(* Logix 5000 project; controller IPG_2332_07A 1769-L16ER-BB1B rev 34.12; software revision 34.01 *)

TASK MAIN_10Ms (periodic, rate 10 ms, priority 1, watchdog 500 ms) : MainProgram_10Ms
TASK MainTask (continuous, watchdog 500 ms) : MainProgram

MODULES
   Local : 1769-L16ER-BB1B (PointIO 0, rev 34.12)
      VS_063 : EX260-SEN1 (Ethernet 192.168.0.63, rev 1.1, Output RPI 10 ms)
      Camera_065 : vendor 678 type 100 code 274 (Ethernet 192.168.0.65, rev 11.1, Output RPI 60 ms)
      QR_064 : vendor 678 type 773 code 1330 (Ethernet 192.168.0.64, rev 1.6, StandardDataDriven RPI 20 ms)
           QR_064:I1.Data[3].4   // QR Results Valid
           QR_064:I1.Data[0].3   // MIssed Trigger
           QR_064:I1.Data[1]   // Results Status
           QR_064:I1.Data[6]   // Trigger Count
           QR_064:I1.Data[1].0   // Results Available
           QR_064:I1.Data[1].7   // General Fault
           QR_064:I1.Data[1].1   // Result Ack Mirror
           QR_064:I1.Data[2].6   // QR Trigger Ack
           QR_064:I1.Data[0].6   // Trigger IN1-Pin4 Current State
           QR_064:I1.Data[0].2   // Aquiring
           QR_064:I1.Data[0].4   // Current Mode (0- Setup Tool Mode, 1- Run Mode)
           QR_064:I1.Data[8]   // Result Count
           QR_064:I1.Data[0].0   // Trigger Ready
           QR_064:I1.Data[0].1   // Trigger Ack
           QR_064:I1.Data[0].5   // Serial Error (0- no error or in configuration mode, 1 - No Reader connected)
           QR_064:I1.Data[1].2   // Result Data Buffer Overrun
           QR_064:I1.Data[0]   // Trigger Status
           QR_064:I1.Data[0].7   // Trigger IN2-Pin2 Current State
           QR_064:O1.Data[0].1   // Trigger
           QR_064:O1.Data[0].0   // Trigger Enable
           QR_064:O1.Data[0].5   // QR Trigger
      Discrete_IO : Embedded (PointIO 1, rev 34.11, Output RPI 20 ms)
      C_ANALOG_01 : 1734-OE2V (PointIO 3, rev 3.1, Output RPI 80 ms)
      RS232 : 1734-232ASC (PointIO 2, rev 4.1, Output RPI 80 ms)
      C_ANALOG_02 : 1734-OE2V (PointIO 4, rev 3.1, Output RPI 80 ms)
END_MODULES

TYPE DateTime :
STRUCT
   Year : DINT;
   Month : DINT;
   Day : DINT;
   Hour : DINT;
   Minute : DINT;
   Second : DINT;
   MicroSecond : DINT;
END_STRUCT
END_TYPE

TYPE String_1 :
STRUCT
   LEN : DINT;
   DATA : SINT[1];
END_STRUCT
END_TYPE

TYPE String_15 :
STRUCT
   LEN : DINT;
   DATA : SINT[15];
END_STRUCT
END_TYPE

TYPE String_60 :
STRUCT
   LEN : DINT;
   DATA : SINT[60];
END_STRUCT
END_TYPE

TYPE udt_Controller_Status :
STRUCT
   Battery_Status : BOOL;
   Forces_Installed : BOOL;
   Forces_Enabled : BOOL;
   Controller_Mode : DINT;   // 1 = Program 2= Run 3 = Remote Run 4= Remote Test 5 = Remote Program 6 = Fault
   Controller_Status : DINT;
   Device_Status : DINT;
   Fault_Status : DINT;
   Forces_Status : DINT;   // 0 = No Forces, Forces not Enabled 1 = Forces Enabled 2 = Forces Installed
   IO_Status : DINT;   // 0 = LED Off 1 = Flashing Red 2 = Flashing Green 3 = Solid Green
   Key_Switch_Status : DINT;   // 1 = Run 2 = Program 3 = Remote
   Minor_Fault : DINT;
END_STRUCT
END_TYPE

TYPE udt_HMI_IO_Desc :
STRUCT
   Increment_Page : BOOL;
   Increment_Event : BOOL;
   Increment_OS : BOOL;
   Decrement_Page : BOOL;
   Decrement_Event : BOOL;
   Decrement_OS : BOOL;
   Two_Column_Display : BOOL;   // On = 2 Column Display
   Index : DINT;
   Max_Index : DINT;   // Maximum Index
   Status : INT[2];
   IO_Desc : udt_IO_Desc[16];
END_STRUCT
END_TYPE

TYPE udt_HMI_Message :
STRUCT
   Message : String_60;
   Background : DINT;
END_STRUCT
END_TYPE

TYPE udt_HMI_Message_Display :
STRUCT
   Message : udt_HMI_Message;
   Index : DINT;
END_STRUCT
END_TYPE

TYPE udt_HMI_Optix :
STRUCT
   Current_Display_Name : STRING;
   Previous_Display_Name : STRING;
   Project_Name : STRING;
   Active_Language : String_15;
   Heartbeat : BOOL;
END_STRUCT
END_TYPE

TYPE udt_HMI_PB :
STRUCT
   PB : DINT;
   ONS : DINT;
   PB_OS : DINT;
END_STRUCT
END_TYPE

TYPE udt_IO_Desc :
STRUCT
   Address : STRING_16;
   Description : STRING_32;
END_STRUCT
END_TYPE

TYPE udt_LED :
STRUCT
   Max_Voltage : INT;
   Ramp_Timer : TIMER;
   On_Timer : TIMER;
   Voltage_Out : INT;
   Delay_Timer : TIMER;
   On_Time : REAL;
   Delay_Time : REAL;
   Ramp_Time : REAL;
END_STRUCT
END_TYPE

TYPE udt_Machine_Control_V2 :
STRUCT
   Alarm : BOOL;
   Alarm_Silence : BOOL;
   Auto_Mode : BOOL;
   Auto_On_OS : BOOL;
   Auto_Off_OS : BOOL;
   Conveyors_Run : BOOL;
   Conveyors_Running : BOOL;
   Conveyors_On_OS : BOOL;
   Conveyors_Off_OS : BOOL;
   Conveyor_Stop_Req : BOOL;
   Conveyor_Stop : BOOL;
   Cycle_Enable : BOOL;   // Cycle Enable
   Fault_Reset : BOOL;   // Reset Fault
   Guard_Closed : BOOL;
   Master_Reset : BOOL;   // Master Reset
   Pwr_Up_Chk : BOOL;   // Power up Light check
   Pwr_On : BOOL;   // Power On
   Reset : BOOL;   // Reset
   Reset_Counts : BOOL;
   Safety_OK : BOOL;   // Safety Ok
   Reset_OS : BOOL;
   Single_Cycle : BOOL;   // Single Cycle
   Single_Cycle_On_OS : BOOL;
   Single_Cycle_Off_OS : BOOL;
   Stop : BOOL;   // Stop Position
   Stop_Pos : BOOL;
   Stop_Req : BOOL;   // Stop Request
   Update_OS : BOOL;   // Update Results
   Start_OS : BOOL;
   Sequence_Reset : BOOL;   // Reset Sequence
   Alarm_Monitor : BOOL[32];   // Alarm Monitor Conditions
   Reset_Cnt : COUNTER;   // Reset Counter
   HMI_Mode_Display : DINT;   // HMI Mode Display
   HMI_PB : udt_HMI_PB;   // HMI Pushbuttons
   Message_Index : DINT;   // MMI Message Index
   OS : DINT;   // one shots
   Counts : DINT[3];   // Station Production Counts
   Conveyor_Start_Dly : TIMER;   // Conveyor Start Delay
   Guard_Close_Delay : TIMER;
   Guard_Unlock_Dly : TIMER;
   Guard_Unlock_Timer : TIMER;
   Pwr_On_Dly : TIMER;   // Power On Delay Timer
   Safety_Ok_Dly : TIMER;   // Safety Ok Delay
   Reset_Duration : TIMER;   // Reset Duration
   Cycle_Time : TIMER;
   Conveyor_Speed : REAL;
END_STRUCT
END_TYPE

TYPE udt_Shift_Register :
STRUCT
   SR : DINT;   // Shift Register
   Part_Style : DINT;   // Part Style
   Height : REAL;   // Height
END_STRUCT
END_TYPE

TYPE udt_Station_Sequence :
STRUCT
   Done : BOOL;   // Sequence Done/Complete
   Home : BOOL;   // Station Home
   In_Process : BOOL;   // Sequence In Process
   Request : BOOL;   // Sequence Request
   Position : DINT;
   OS : DINT;
   OS1 : DINT;
   OS2 : DINT;
   StepOS : DINT;
   StepOS1 : DINT;
   StepOS2 : DINT;
   Timer : TIMER[20];
   Result : BOOL;   // 0=Fail, 1=Pass
END_STRUCT
END_TYPE

TYPE udt_Zaber_Axis :
STRUCT
   Home : BOOL;
   InPos : BOOL;
   ActPos_Step_String : STRING;
   CmdPos_mm : REAL;
   CmdPos_Step_Dint : DINT;
   CmdPos_Step_String : STRING;
   Write_String : STRING;
   Read_String : STRING;
   Write : SERIAL_PORT_CONTROL;
   MoveReq : BOOL;
   Reset : BOOL;
   Home_String : STRING; {access Read Only}
   MovAbs_String : STRING;
   MovAbs : BOOL;
   Return_String : STRING;
   MovRel_String : STRING;
   MovRel : BOOL;
   Resloution : REAL;   // micrometers per step
   Manual_MovAbs : BOOL;
   Jog_Fwd : BOOL;
   Jog_Fwd_String : STRING;
   Jog_Rev : BOOL;
   Jog_Rev_String : STRING;
   Jog_Value_mm : REAL;
   Go_Home : BOOL;
   Go_CmdPos : BOOL;
   Jog_Value_Step_Dint : DINT;
   Jog_Value_Step_String : STRING;
   Store_CmdPos : BOOL;
   Get_Pos_String : STRING;
   Store_CmdPos_Delay : TIMER;
   String_Pos_Found : DINT;
   String_Pos_Length : DINT;
   Get_Pos : BOOL;
   WriteReq : BOOL;
   Status : STRING;
   Moving : BOOL;
   Idle : STRING;
   IdlePos : DINT;
   Zero : STRING;
   Get_Pos_Delay : TIMER;
   Busy : STRING;
   BusyPos : DINT;
   Axis_String : STRING;
   Axis_Dint : DINT;
   HMI_PB : udt_HMI_PB;
   Store_CmdPos_Reset_Delay : TIMER;
   ActPos_Step_Dint : DINT;
   ActPos_mm : REAL;
   Reset_String : STRING;
END_STRUCT
END_TYPE

ADD_ON_INSTRUCTION AOI_Convert_hhmmss   (* revision 1.0 *)
VAR_INPUT
   Hour : DINT; {required}
   Minutes : DINT; {required}
   Seconds : DINT; {required}
END_VAR
VAR_IN_OUT
   Time : String_15; {required}
END_VAR
VAR
   String_Hour : String_15; {access None}
   String_Minute : String_15; {access None}
   String_Seconds : String_15; {access None}
   String_Colon : String_1 := ':'; {access None}
   Temp_String : String_15; {access None}
   String_Zero : String_1 := '0'; {access None}
END_VAR

ROUTINE Logic   (* ladder *)
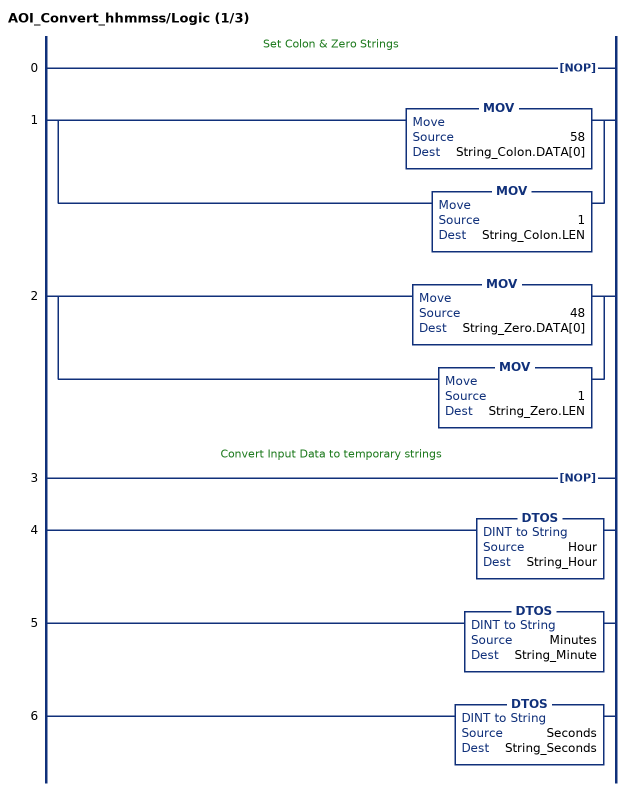
   // Set Colon & Zero Strings
   0: NOP();
   1: [MOV(58,String_Colon.DATA[0]) ,MOV(1,String_Colon.LEN) ];
   2: [MOV(48,String_Zero.DATA[0]) ,MOV(1,String_Zero.LEN) ];
   // Convert Input Data to temporary strings
   3: NOP();
   4: DTOS(Hour,String_Hour);
   5: DTOS(Minutes,String_Minute);
   6: DTOS(Seconds,String_Seconds);
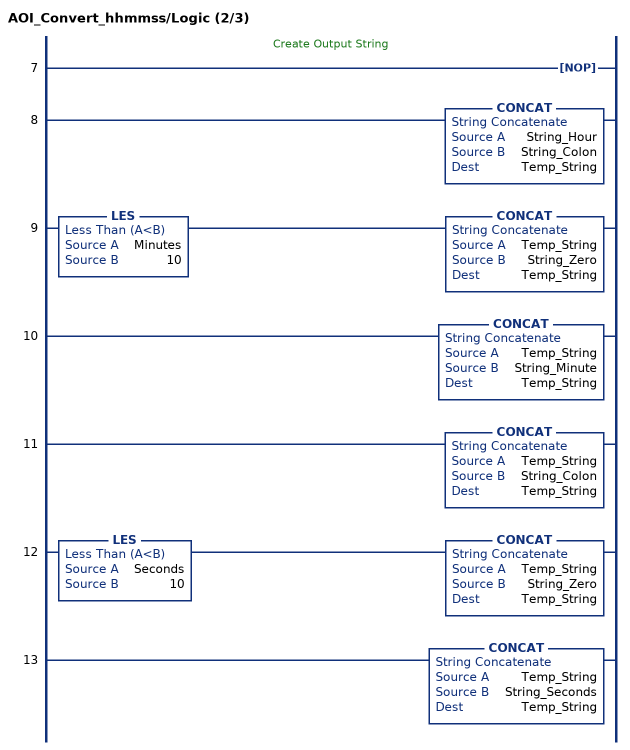
   // Create Output String
   7: NOP();
   8: CONCAT(String_Hour,String_Colon,Temp_String);
   9: LES(Minutes,10)CONCAT(Temp_String,String_Zero,Temp_String);
   10: CONCAT(Temp_String,String_Minute,Temp_String);
   11: CONCAT(Temp_String,String_Colon,Temp_String);
   12: LES(Seconds,10)CONCAT(Temp_String,String_Zero,Temp_String);
   13: CONCAT(Temp_String,String_Seconds,Temp_String);
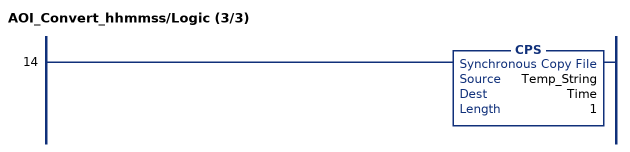
   14: CPS(Temp_String,Time,1);
END_ROUTINE
END_ADD_ON_INSTRUCTION

ADD_ON_INSTRUCTION AOI_Cycle_Times   (* revision 1.0 *)
VAR_INPUT
   Start_Timing_IN : BOOL; {visible}
   In_Process_IN : BOOL; {visible}
   Alarmed_IN : BOOL; {visible}
   Waiting_IN : BOOL; {visible}
   Update_IN : BOOL; {visible}
   Uptime_IN : BOOL; {visible}
   Downtime_IN : BOOL; {visible}
   Data_Reset_IN : BOOL; {visible}
END_VAR
VAR_OUTPUT
   Avg_Cycle_Time : REAL; {access Read Only, visible}
   Cycle_Time : REAL; {access Read Only, visible}
   Avg_PTP_Cycle_Time : REAL; {access Read Only, visible}
   Part_Part_Cycle_Time : REAL; {access Read Only, visible}
END_VAR
VAR_INPUT
   Current_Cycle : REAL; {visible}
END_VAR
VAR_IN_OUT
   Waiting_Time : String_15; {required}
   Alarmed_Time : String_15; {required}
   Uptime_Time : String_15; {required}
   Downtime_Time : String_15; {required}
END_VAR
VAR
   p_Timer : TIMER := (PRE := 100); {access None}
   p_Accumulated_mS : DINT; {access None}
   p_ONS : DINT; {access None}
   p_Start_Time_mS : DINT; {access None}
   p_End_Time_mS : DINT; {access None}
   p_Cycle_Time_mS : DINT; {access None}
   p_Total_Cycles : DINT; {access None}
   p_Avg_PTP_Cycle_Time_Raw : DINT; {access None}
   p_Waiting_Accumulated_mS : DINT; {access None}
   p_Convert_Waiting_AOI : AOI_Convert_hhmmss; {access None}
   p_Convert_Alarmed_AOI : AOI_Convert_hhmmss; {access None}
   p_Avg_Cycle_Time_Raw : DINT; {access None}
   p_Uptime_mSeconds : DINT; {access None}
   p_Uptime_Seconds : DINT; {access None}
   p_Uptime_Minutes : DINT; {access None}
   p_Uptime_Hours : DINT; {access None}
   p_Convert_Uptime_AOI : AOI_Convert_hhmmss; {access None}
   p_Waiting_Hours : DINT; {access Read Only}
   p_Waiting_Minutes : DINT; {access Read Only}
   p_Waiting_Seconds : DINT; {access Read Only}
   p_Alarm_Hours : DINT; {access Read Only}
   p_Alarm_Minutes : DINT; {access Read Only}
   p_Alarm_mSeconds : DINT; {access None}
   p_Alarm_Seconds : DINT; {access Read Only}
   p_Convert_Downtime_AOI : AOI_Convert_hhmmss; {access None}
   p_Downtime_Hours : DINT; {access None}
   p_Downtime_Minutes : DINT; {access None}
   p_Downtime_Seconds : DINT; {access None}
   p_Downtime_mSeconds : DINT; {access None}
END_VAR

ROUTINE Logic   (* ladder *)
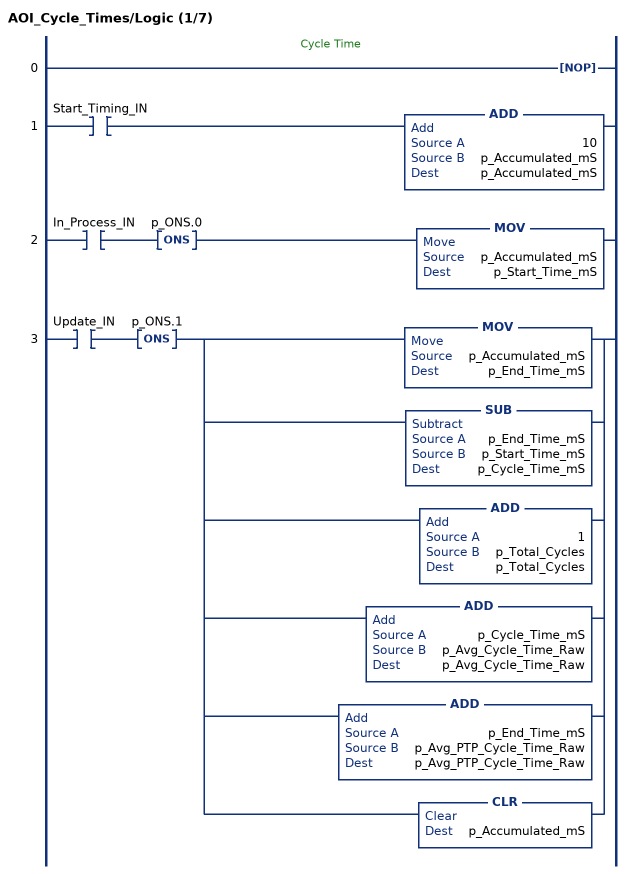
   // Cycle Time
   0: NOP();
   1: XIC(Start_Timing_IN)ADD(10,p_Accumulated_mS,p_Accumulated_mS);
   2: XIC(In_Process_IN)ONS(p_ONS.0)MOV(p_Accumulated_mS,p_Start_Time_mS);
   3: XIC(Update_IN)ONS(p_ONS.1)[MOV(p_Accumulated_mS,p_End_Time_mS) ,SUB(p_End_Time_mS,p_Start_Time_mS,p_Cycle_Time_mS) ,ADD(1,p_Total_Cycles,p_Total_Cycles) ,ADD(p_Cycle_Time_mS,p_Avg_Cycle_Time_Raw,p_Avg_Cycle_Time_Raw) ,ADD(p_End_Time_mS,p_Avg_PTP_Cycle_Time_Raw,p_Avg_PTP_Cycle_Time_Raw) ,CLR(p_Accumulated_mS) ];
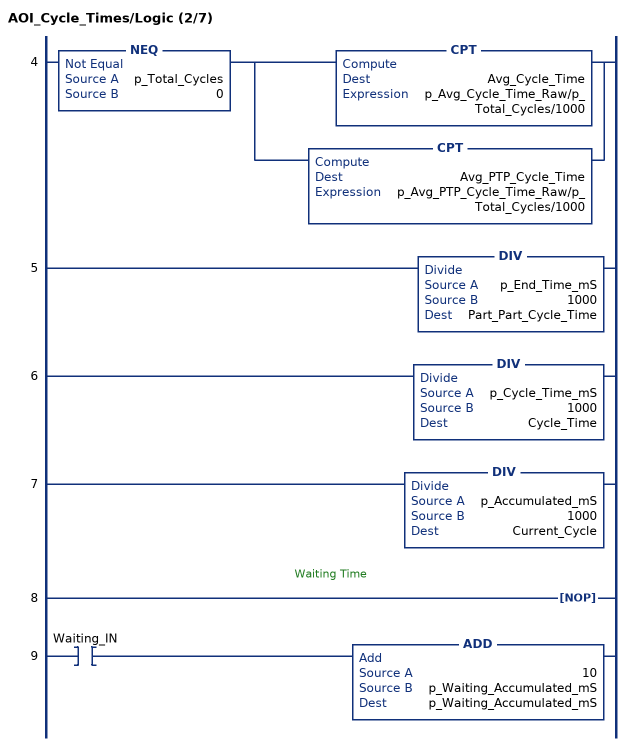
   4: NEQ(p_Total_Cycles,0)[CPT(Avg_Cycle_Time,p_Avg_Cycle_Time_Raw/p_Total_Cycles/1000) ,CPT(Avg_PTP_Cycle_Time,p_Avg_PTP_Cycle_Time_Raw/p_Total_Cycles/1000) ];
   5: DIV(p_End_Time_mS,1000,Part_Part_Cycle_Time);
   6: DIV(p_Cycle_Time_mS,1000,Cycle_Time);
   7: DIV(p_Accumulated_mS,1000,Current_Cycle);
   // Waiting Time
   8: NOP();
   9: XIC(Waiting_IN)ADD(10,p_Waiting_Accumulated_mS,p_Waiting_Accumulated_mS);
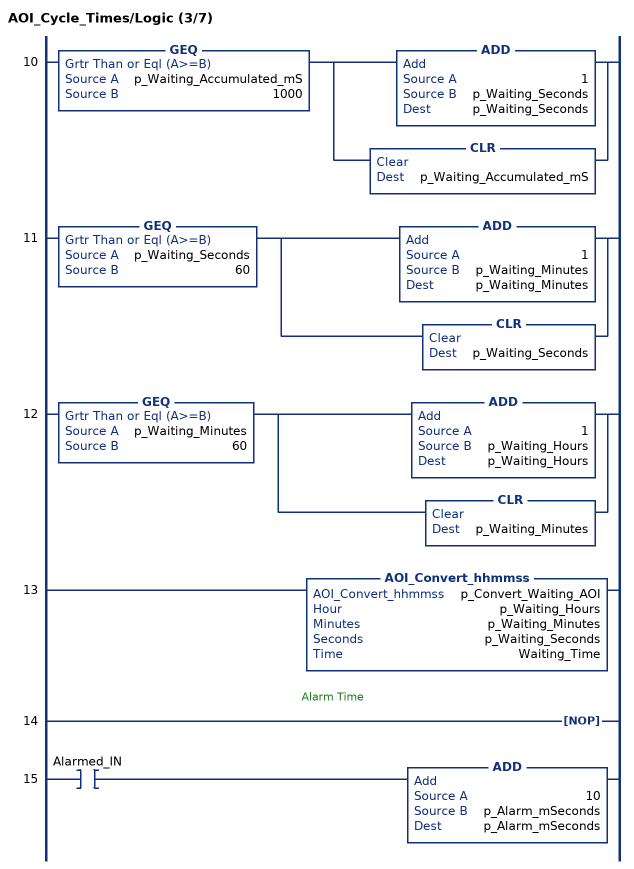
   10: GEQ(p_Waiting_Accumulated_mS,1000)[ADD(1,p_Waiting_Seconds,p_Waiting_Seconds) ,CLR(p_Waiting_Accumulated_mS) ];
   11: GEQ(p_Waiting_Seconds,60)[ADD(1,p_Waiting_Minutes,p_Waiting_Minutes) ,CLR(p_Waiting_Seconds) ];
   12: GEQ(p_Waiting_Minutes,60)[ADD(1,p_Waiting_Hours,p_Waiting_Hours) ,CLR(p_Waiting_Minutes) ];
   13: AOI_Convert_hhmmss(p_Convert_Waiting_AOI,p_Waiting_Hours,p_Waiting_Minutes,p_Waiting_Seconds,Waiting_Time);
   // Alarm Time
   14: NOP();
   15: XIC(Alarmed_IN)ADD(10,p_Alarm_mSeconds,p_Alarm_mSeconds);
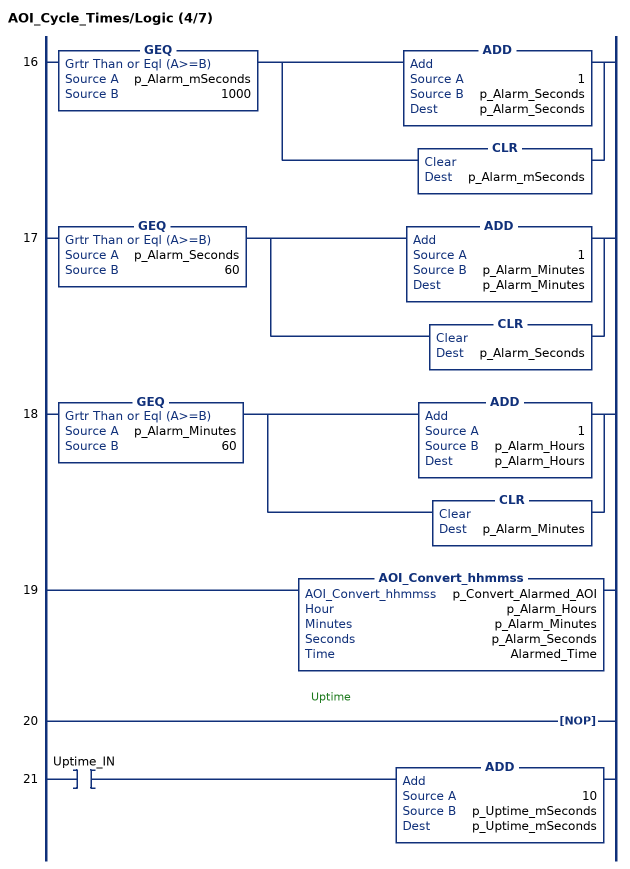
   16: GEQ(p_Alarm_mSeconds,1000)[ADD(1,p_Alarm_Seconds,p_Alarm_Seconds) ,CLR(p_Alarm_mSeconds) ];
   17: GEQ(p_Alarm_Seconds,60)[ADD(1,p_Alarm_Minutes,p_Alarm_Minutes) ,CLR(p_Alarm_Seconds) ];
   18: GEQ(p_Alarm_Minutes,60)[ADD(1,p_Alarm_Hours,p_Alarm_Hours) ,CLR(p_Alarm_Minutes) ];
   19: AOI_Convert_hhmmss(p_Convert_Alarmed_AOI,p_Alarm_Hours,p_Alarm_Minutes,p_Alarm_Seconds,Alarmed_Time);
   // Uptime
   20: NOP();
   21: XIC(Uptime_IN)ADD(10,p_Uptime_mSeconds,p_Uptime_mSeconds);
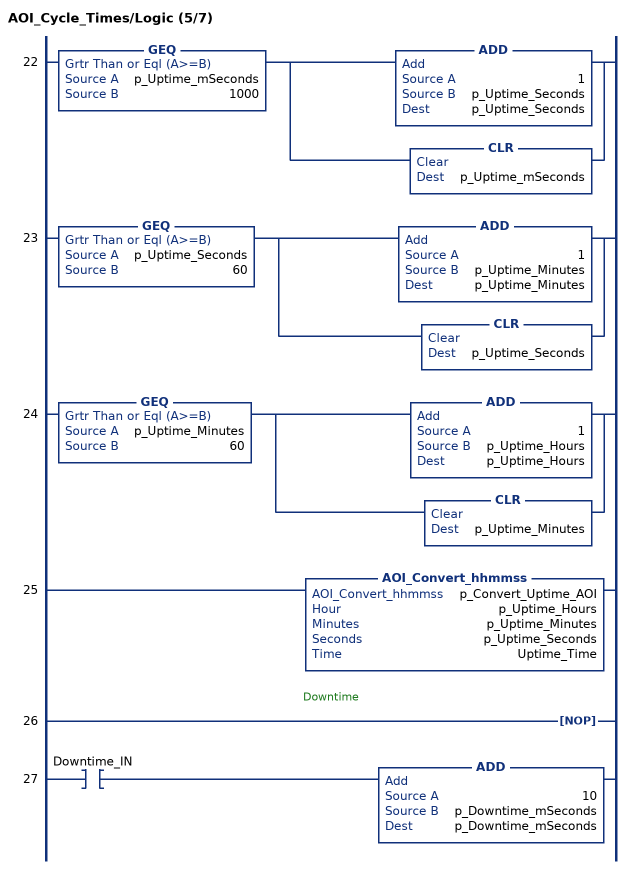
   22: GEQ(p_Uptime_mSeconds,1000)[ADD(1,p_Uptime_Seconds,p_Uptime_Seconds) ,CLR(p_Uptime_mSeconds) ];
   23: GEQ(p_Uptime_Seconds,60)[ADD(1,p_Uptime_Minutes,p_Uptime_Minutes) ,CLR(p_Uptime_Seconds) ];
   24: GEQ(p_Uptime_Minutes,60)[ADD(1,p_Uptime_Hours,p_Uptime_Hours) ,CLR(p_Uptime_Minutes) ];
   25: AOI_Convert_hhmmss(p_Convert_Uptime_AOI,p_Uptime_Hours,p_Uptime_Minutes,p_Uptime_Seconds,Uptime_Time);
   // Downtime
   26: NOP();
   27: XIC(Downtime_IN)ADD(10,p_Downtime_mSeconds,p_Downtime_mSeconds);
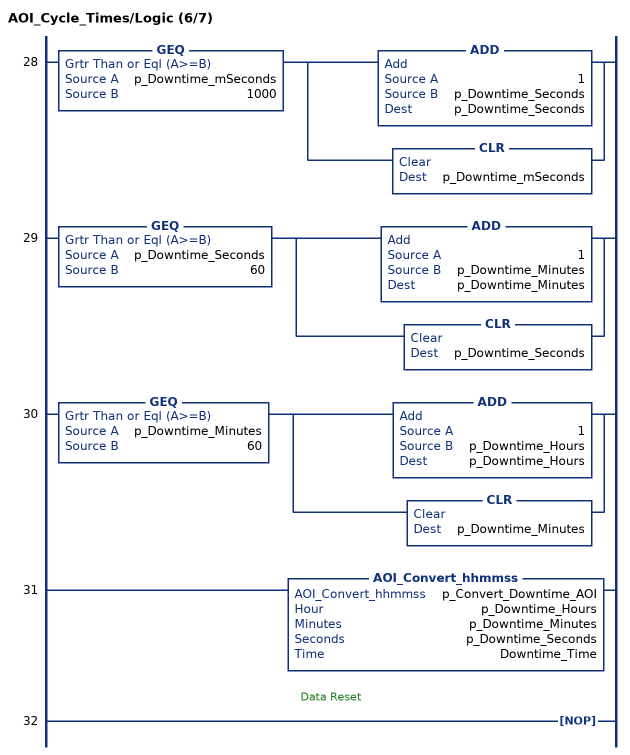
   28: GEQ(p_Downtime_mSeconds,1000)[ADD(1,p_Downtime_Seconds,p_Downtime_Seconds) ,CLR(p_Downtime_mSeconds) ];
   29: GEQ(p_Downtime_Seconds,60)[ADD(1,p_Downtime_Minutes,p_Downtime_Minutes) ,CLR(p_Downtime_Seconds) ];
   30: GEQ(p_Downtime_Minutes,60)[ADD(1,p_Downtime_Hours,p_Downtime_Hours) ,CLR(p_Downtime_Minutes) ];
   31: AOI_Convert_hhmmss(p_Convert_Downtime_AOI,p_Downtime_Hours,p_Downtime_Minutes,p_Downtime_Seconds,Downtime_Time);
   // Data Reset
   32: NOP();
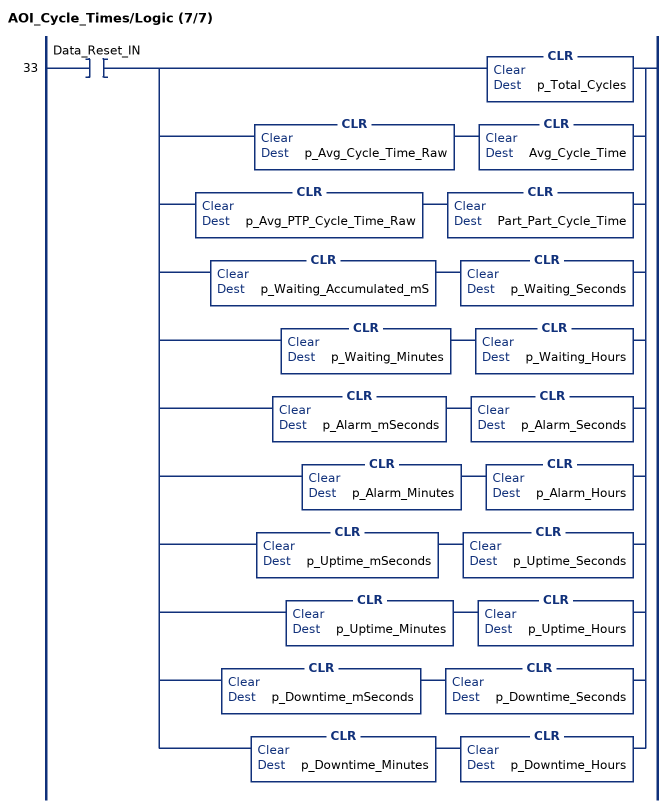
   33: XIC(Data_Reset_IN)[CLR(p_Total_Cycles) ,CLR(p_Avg_Cycle_Time_Raw) CLR(Avg_Cycle_Time) ,CLR(p_Avg_PTP_Cycle_Time_Raw) CLR(Part_Part_Cycle_Time) ,CLR(p_Waiting_Accumulated_mS) CLR(p_Waiting_Seconds) ,CLR(p_Waiting_Minutes) CLR(p_Waiting_Hours) ,CLR(p_Alarm_mSeconds) CLR(p_Alarm_Seconds) ,CLR(p_Alarm_Minutes) CLR(p_Alarm_Hours) ,CLR(p_Uptime_mSeconds) CLR(p_Uptime_Seconds) ,CLR(p_Uptime_Minutes) CLR(p_Uptime_Hours) ,CLR(p_Downtime_mSeconds) CLR(p_Downtime_Seconds) ,CLR(p_Downtime_Minutes) CLR(p_Downtime_Hours) ];
END_ROUTINE
END_ADD_ON_INSTRUCTION

ADD_ON_INSTRUCTION AOI_PB_Confirm   (* revision 1.0 *)
VAR_INPUT
   Pushbutton_IN : BOOL; {required}
END_VAR
VAR_OUTPUT
   Confirmed_OUT : BOOL; {access Read Only, visible}
   State_OUT : DINT; {access Read Only, visible}
END_VAR
VAR
   PB_ONS : BOOL; {access None}
   Confirm_CTU : COUNTER := (PRE := 2); {access None}
   Confirm_Timeout : TIMER := (PRE := 2000); {access None}
   Confirmed_ONS : BOOL; {access None}
END_VAR

ROUTINE Logic   (* ladder *)
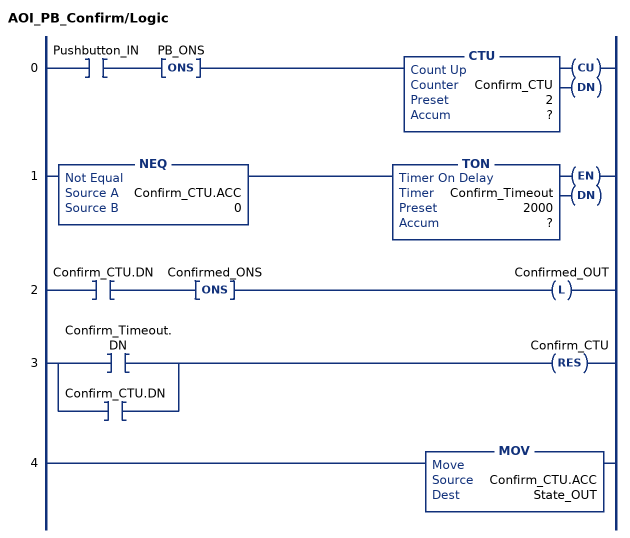
   0: XIC(Pushbutton_IN)ONS(PB_ONS)CTU(Confirm_CTU,?,?);
   1: NEQ(Confirm_CTU.ACC,0)TON(Confirm_Timeout,?,?);
   2: XIC(Confirm_CTU.DN)ONS(Confirmed_ONS)OTL(Confirmed_OUT);
   3: [XIC(Confirm_Timeout.DN) ,XIC(Confirm_CTU.DN) ]RES(Confirm_CTU);
   4: MOV(Confirm_CTU.ACC,State_OUT);
END_ROUTINE
END_ADD_ON_INSTRUCTION

ADD_ON_INSTRUCTION AOI_PLC_Status   (* revision 1.0 *)
VAR_IN_OUT
   HMI_PLC_Status : udt_Controller_Status; {required}
END_VAR

ROUTINE Logic   (* ladder *)
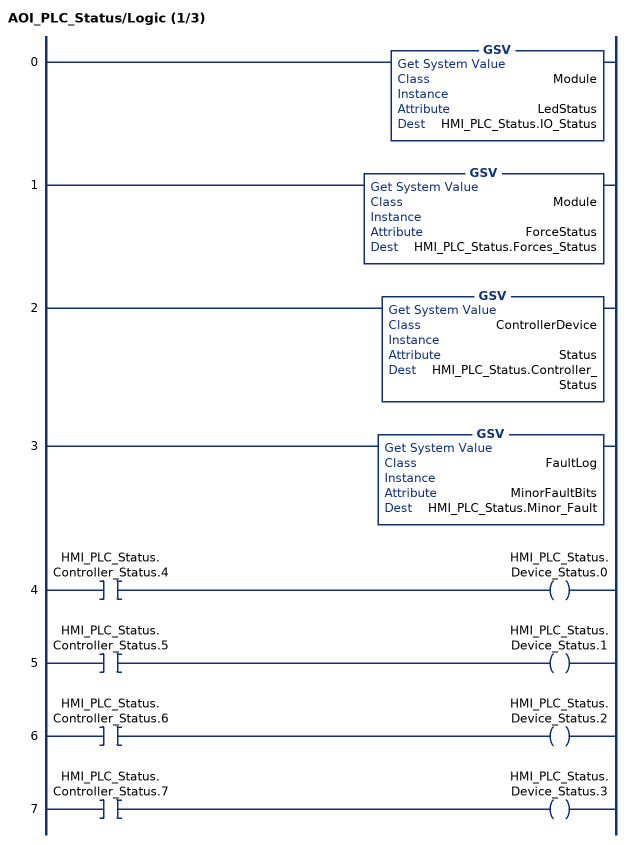
   0: GSV(Module,,LedStatus,HMI_PLC_Status.IO_Status);
   1: GSV(Module,,ForceStatus,HMI_PLC_Status.Forces_Status);
   2: GSV(ControllerDevice,,Status,HMI_PLC_Status.Controller_Status);
   3: GSV(FaultLog,,MinorFaultBits,HMI_PLC_Status.Minor_Fault);
   4: XIC(HMI_PLC_Status.Controller_Status.4)OTE(HMI_PLC_Status.Device_Status.0);
   5: XIC(HMI_PLC_Status.Controller_Status.5)OTE(HMI_PLC_Status.Device_Status.1);
   6: XIC(HMI_PLC_Status.Controller_Status.6)OTE(HMI_PLC_Status.Device_Status.2);
   7: XIC(HMI_PLC_Status.Controller_Status.7)OTE(HMI_PLC_Status.Device_Status.3);
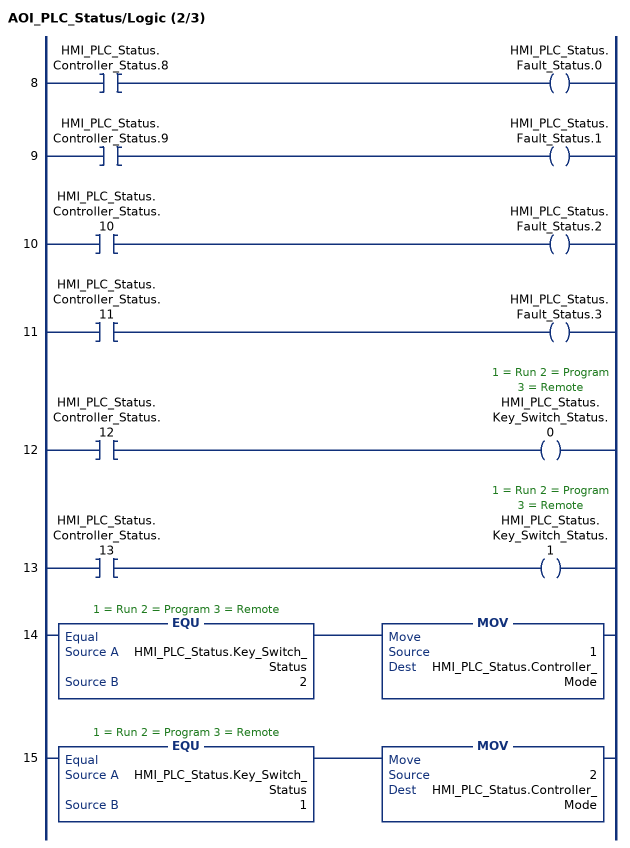
   8: XIC(HMI_PLC_Status.Controller_Status.8)OTE(HMI_PLC_Status.Fault_Status.0);
   9: XIC(HMI_PLC_Status.Controller_Status.9)OTE(HMI_PLC_Status.Fault_Status.1);
   10: XIC(HMI_PLC_Status.Controller_Status.10)OTE(HMI_PLC_Status.Fault_Status.2);
   11: XIC(HMI_PLC_Status.Controller_Status.11)OTE(HMI_PLC_Status.Fault_Status.3);
   12: XIC(HMI_PLC_Status.Controller_Status.12)OTE(HMI_PLC_Status.Key_Switch_Status.0);
   13: XIC(HMI_PLC_Status.Controller_Status.13)OTE(HMI_PLC_Status.Key_Switch_Status.1);
   14: EQU(HMI_PLC_Status.Key_Switch_Status,2)MOV(1,HMI_PLC_Status.Controller_Mode);
   15: EQU(HMI_PLC_Status.Key_Switch_Status,1)MOV(2,HMI_PLC_Status.Controller_Mode);
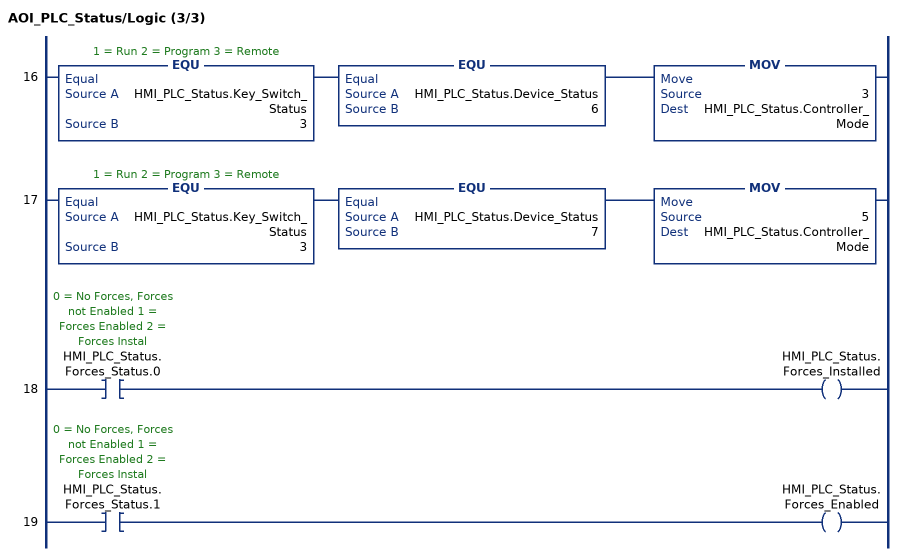
   16: EQU(HMI_PLC_Status.Key_Switch_Status,3)EQU(HMI_PLC_Status.Device_Status,6)MOV(3,HMI_PLC_Status.Controller_Mode);
   17: EQU(HMI_PLC_Status.Key_Switch_Status,3)EQU(HMI_PLC_Status.Device_Status,7)MOV(5,HMI_PLC_Status.Controller_Mode);
   18: XIC(HMI_PLC_Status.Forces_Status.0)OTE(HMI_PLC_Status.Forces_Installed);
   19: XIC(HMI_PLC_Status.Forces_Status.1)OTE(HMI_PLC_Status.Forces_Enabled);
END_ROUTINE
END_ADD_ON_INSTRUCTION

VAR_GLOBAL   (* controller tags *)
   DateTime : DateTime := (Year := 2023, Month := 12, Day := 8, Hour := 12, Minute := 11, Second := 26, MicroSecond := 594656);
   Debug_SDF : DINT := 64;
   HMI_IO_Description : udt_IO_Desc[96] := ([0].Address := 'Loc:I:1.0', [0].Description := 'E-Stop Relay Monitor', [1].Address := 'Loc:I:1.1', [1].Description := 'E-Stop PB', [2].Address := 'Loc:I:1.2', [2].Description := 'Door Safety Relay Monitor', [3].Address := 'Loc:I:1.3', [3].Description := 'Main Air Okay', [4].Address := 'Loc:I:1.4', [4].Description := 'Start PB', [5].Address := 'Loc:I:1.5', [5].Description := 'Spare', [6].Address := 'Loc:I:1.6', [6].Description := 'Spare', [7].Address := 'Loc:I:1.7', [7].Description := 'Spare', [8].Address := 'Loc:I:1.8', [8].Description := 'Ferrule Gripper Vac', [9].Address := 'Loc:I:1.9', [9].Description := 'Fiber Gripper Vac', [10].Address := 'Loc:I:1.10', [10].Description := 'Cassette Gripper Release', [11].Address := 'Loc:I:1.11', [11].Description := 'Cassette Gripper Extend', [12].Address := 'Loc:I:1.12', [12].Description := 'Cassette Gripper Retract', [13].Address := 'Loc:I:1.13', [13].Description := 'Cassette Presence', [14].Address := 'Loc:I:1.14', [14].Description := 'Spare', [15].Address := 'Loc:I:1.15', [15].Description := 'Spare', [16].Address := 'Loc:O:1.0', [16].Description := 'E-Stop Safety Reset', [17].Address := 'Loc:O:1.1', [17].Description := 'Spare', [18].Address := 'Loc:O:1.2', [18].Description := 'Light Stack Read', [19].Address := 'Loc:O:1.3', [19].Description := 'Light Stack Amber', [20].Address := 'Loc:O:1.4', [20].Description := 'Light Stack Green', [21].Address := 'Loc:O:1.5', [21].Description := 'Ferrule Gripper Solenoid', [22].Address := 'Loc:O:1.6', [22].Description := 'Fiber Gripper Solenoid', [23].Address := 'Loc:O:1.7', [23].Description := 'Spare', [24].Address := 'Loc:O:1.8', [24].Description := 'Dispenser Start', [25].Address := 'Loc:O:1.9', [25].Description := 'PB Light Red', [26].Address := 'Loc:O:1.10', [26].Description := 'PB Light Amber', [27].Address := 'Loc:O:1.11', [27].Description := 'PB Light Green', [28].Address := 'Loc:O:1.12', [28].Description := 'Work Light', [29].Address := 'Loc:O:1.13', [29].Description := 'Spare',
        [30].Address := 'Loc:O:1.14', [30].Description := 'Spare', [31].Address := 'Loc:O:1.15', [31].Description := 'Spare', [32].Address := 'VS_063:O:0.0', [32].Description := 'Cassette Release');
   HMI_Messages : udt_HMI_Message_Display[48] := ([1].Message.Message := 'Emergency Stop', [1].Message.Background := 1, [2].Message.Background := 1, [3].Message.Background := 1, [4].Message.Background := 1, [5].Message.Background := 1, [6].Message.Background := 1, [7].Message.Background := 1, [8].Message.Background := 1, [9].Message.Background := 1, [10].Message.Background := 1, [11].Message.Background := 1, [12].Message.Background := 1, [13].Message.Background := 1, [14].Message.Background := 1, [15].Message.Background := 1, [16].Message.Message := 'Safety Reset Required', [16].Message.Background := 6, [17].Message.Message := 'Machine Powering Up', [17].Message.Background := 4, [18].Message.Background := 4, [19].Message.Background := 3, [20].Message.Background := 3, [21].Message.Background := 3, [22].Message.Background := 3, [23].Message.Background := 3, [24].Message.Background := 3, [25].Message.Background := 3, [26].Message.Background := 3, [27].Message.Background := 3, [28].Message.Background := 3, [29].Message.Background := 3, [30].Message.Background := 3, [35].Message.Message := 'Machine Idle', [36].Message.Message := 'Machine Alarmed', [36].Message.Background := 1, [37].Message.Message := 'Machine Running', [37].Message.Background := 2, [41].Message.Message := 'Machine Stop Requested', [41].Message.Background := 2, [42].Message.Message := 'Machine in Setup/Step Mode', [42].Message.Background := 4, [44].Message.Message := 'Cycle Stop in Progress');
   HMI_Messages_Sequence : udt_HMI_Message_Display[20] := ([0].Message.Message := 'Idle', [1].Message.Message := 'Waiting for Cassette', [1].Message.Background := 4, [2].Message.Message := 'Fiber Vacuum On', [2].Message.Background := 2, [3].Message.Message := 'Ferrule Vacuum On', [3].Message.Background := 2, [4].Message.Message := 'Read Database', [4].Message.Background := 2, [5].Message.Message := 'Check Database', [5].Message.Background := 2, [6].Message.Message := 'Fiber Axis Down', [6].Message.Background := 2, [7].Message.Message := 'Syringe Axis In', [7].Message.Background := 2, [8].Message.Message := 'Dispense Glue', [8].Message.Background := 2, [9].Message.Message := 'Syringe Axis Out', [9].Message.Background := 2, [10].Message.Message := 'Mirror Axis In', [10].Message.Background := 2, [11].Message.Message := 'LED On', [11].Message.Background := 2, [12].Message.Message := 'Mirror Axis Out', [12].Message.Background := 2, [13].Message.Message := 'Ferrule Vacuum Off', [13].Message.Background := 2, [14].Message.Message := 'Fiber Axis Up', [14].Message.Background := 2, [15].Message.Message := 'Fiber Vacuum Off', [15].Message.Background := 2, [16].Message.Message := 'Sequence Complete', [16].Message.Background := 2, [17].Message.Background := 2, [18].Message.Background := 2, [19].Message.Background := 2);
END_VAR

PROGRAM MainProgram   (* main routine MainRoutine *)

ROUTINE MainRoutine   (* ladder *)
END_ROUTINE
END_PROGRAM

PROGRAM MainProgram_10Ms   (* main routine A_Main *)
VAR
   Axis_Controller : udt_Zaber_Axis := (Write_String := '/1 3 get pos$0D', Read_String := '$0A@01 3 OK IDLE -- 0$0D', Write.LEN := -243409016, Write.POS := -2147483640, Write.ERROR := 16#8000_0008, Home_String := '$C1$00$1C$00$01$00$00$00$00$00$00$00$00$00$00$00$08$00$00$80L$00$00$80$CCt9$F1$04<$00$00$9C$84$1B$00$14$01$00$00$02$00$00$00$00$00$00$00$01$00$00$00$00$00$00$00$00$00$00$00$00$00$00$00$00$00$00$00$00$00$00$00$00$00$00$00$00$00$00$00$00$00$00$00', Resloution := 8.e-45, Manual_MovAbs := 1, Jog_Rev_String := ' ', Go_CmdPos := 1, Jog_Value_Step_Dint := 32, Get_Pos_String := '$01$00$00$00$00$00$00$00$00$00$00$00$08$00$00$80$08$00$00$80$CCt9$F1$8C>$00$00$C1$00$15$00$01$00$00$00$00$00$00$00$18$00$08$80$08$00$00$80$08$00$00$80$CCt9$F1$AC>$00$00$C1$00$14$00$01$00$00$00$00$00$00$00$F4$01$00$00$08$00$00$80$08$00$00$80', Store_CmdPos_Delay.PRE := 16076, Store_CmdPos_Delay.ACC := 1245377, Store_CmdPos_Delay.EN := 1, Store_CmdPos_Delay.TT := 1, Store_CmdPos_Delay.DN := 1, String_Pos_Found := 1, Status := '$08$00$00$80$CCt9$F1$EC>$00$00$C1$00$12$00$01$00$00$00$00$00$00$00$00$00$00$00$08$00$00$80$08$00$00$80$CCt9$F1$0C?$00$00$C1$00$11$00$01$00$00$00$00$00$00$00$00$00$00$00$08$00$00$80$08$00$00$80$CCt9$F1,?$00$00$C1$00$10$00$01$00$00$00', Idle := 'IDLE', IdlePos := 1, Get_Pos_Delay.PRE := 1, Busy := 'BUSY', BusyPos := 1, Axis_String := '3', Axis_Dint := 3, HMI_PB.PB := 1, HMI_PB.ONS := 1, Store_CmdPos_Reset_Delay.PRE := -2147483640, Store_CmdPos_Reset_Delay.ACC := -247892788, Store_CmdPos_Reset_Delay.EN := 1, ActPos_Step_Dint := 16588, ActPos_mm := 2.75777e-40);
   Flash_1280mS : BOOL := 1;
   Flash_320mS : BOOL := 1;
   Flash_640mS : BOOL := 1;
   p_Alarmed_Time : String_15 := '0:00:00';
   p_All_Axis_Home : DINT;
        .0   // Home All Req
        .1   // Home Fiber Axis
        .2   // Home Syringe Axis
        .3   // Home Mirror Axis
   p_ALMD_00 : ALARM_DIGITAL;
   p_ALMD_01 : ALARM_DIGITAL;
   p_ALMD_02 : ALARM_DIGITAL;
   p_ALMD_03 : ALARM_DIGITAL;
   p_ALMD_04 : ALARM_DIGITAL;
   p_ALMD_05 : ALARM_DIGITAL;
   p_AOI_Cycle_Times : AOI_Cycle_Times := (Downtime_IN := 1, Data_Reset_IN := 1);
   p_AOI_PLC_Status : AOI_PLC_Status;
   p_ASCII_RXID : DINT := -9;
   p_ASCII_TXID : COUNTER := (ACC := 186, DN := 1);
   p_Axis_ONS : DINT := 256;
   p_Barcode_results_Count_prev : DINT := 2;
   p_Barcode_Results_Ready : BOOL := 1;
   p_BarcodeDone : BOOL;
   p_Cassette_Data : DINT;
   p_Cassette_Data_String : STRING := '000000';
   p_CassetteGripper_Ext_IN : BOOL;
   p_CassetteGripper_OUT : BOOL;
   p_CassetteGripper_Ret_IN : BOOL;
   p_CassettePresence_IN : BOOL;
   p_CassetteRelease_IN : BOOL;   // Foot Switch
   p_Control : udt_Machine_Control_V2 := (Alarm_Silence := 1, Pwr_On := 1, Safety_OK := 1, Message_Index := -247892788, OS := 4312, Counts[0] := 3154114, Counts[1] := 1, Counts[2] := 32, Guard_Unlock_Timer.PRE := -2147483640, Guard_Unlock_Timer.ACC := -247892788, Guard_Unlock_Timer.EN := 1, Pwr_On_Dly.PRE := 500, Pwr_On_Dly.ACC := 500, Pwr_On_Dly.EN := 1, Pwr_On_Dly.DN := 1, Safety_Ok_Dly.PRE := 500, Safety_Ok_Dly.ACC := 500, Safety_Ok_Dly.EN := 1, Safety_Ok_Dly.DN := 1, Reset_Duration.PRE := 2000, Cycle_Time.PRE := 32);   // Main Control
        .OS   // Main Control One Shots
        .HMI_PB.PB.5   // Cycle Step PB
        .HMI_PB.PB_OS.5   // Cycle Step PB OS
   p_Data_Reset : BOOL := 1;
   p_DispenseStart_OUT : BOOL;
   p_DispenseTime : REAL;
   p_DoorMonitor_IN : BOOL;
   p_Downtime : String_15 := '0:00:00';
   p_EstopMonitor_IN : BOOL;
   p_EStopPB_IN : BOOL;
   p_EstopReset_OUT : BOOL;
   p_FerruleGripper_IN : BOOL;
   p_FerruleGripper_OUT : BOOL;
   p_FiberAxis : udt_Zaber_Axis := (Home := 1, ActPos_Step_String := '0', CmdPos_mm := 40.00004, CmdPos_Step_Dint := 403150, CmdPos_Step_String := '403150', Home_String := '/1 1 home$0D', MovAbs_String := '/1 1 move abs ', Return_String := '$0D', MovRel_String := '/1 1 mov rel -', Resloution := 0.09921875, Jog_Fwd_String := '/1 1 move rel  ', Jog_Rev_String := '/1 1 move rel  -', Jog_Value_mm := 0.05, Jog_Value_Step_Dint := 504, Jog_Value_Step_String := '504', Get_Pos_String := '/1 1 get pos$0D', Store_CmdPos_Delay.PRE := 1000, String_Pos_Found := 20, String_Pos_Length := 1, IdlePos := 11, Zero := '0', Get_Pos_Delay.PRE := 1000, Store_CmdPos_Reset_Delay.PRE := 1500);
        .HMI_PB.PB_OS.4   // Go Home
        .HMI_PB.PB.2   // Jog Rev
        .HMI_PB.PB.3   // Jog Fwd
        .HMI_PB.PB.4   // Go Home
        .HMI_PB.PB_OS.2   // Jog Rev
        .HMI_PB.PB_OS.3   // Jog Fwd
        .HMI_PB.PB_OS.0   // Go Cmd Position
        .HMI_PB.PB.1   // Store Cmd Position
        .HMI_PB.PB_OS.1   // Store Cmd Position
        .HMI_PB.PB.0   // Go Cmd Position
   p_FiberAxis_AdjPos : STRING;
   p_FiberAxis_FinalMove_Done : BOOL := 1;
   p_FiberAxis_FinalMoveRel : BOOL;
   p_FiberAxis_FindPos : udt_Station_Sequence := (OS := 1);
   p_FiberAxis_InitialMove_Done : BOOL;
   p_FiberAxis_InitialMoveRel : BOOL;
   p_FiberAxis_Move_01 : DINT := 10; {constant}
   p_FiberAxis_Move_01_String : STRING := '10';
   p_FiberAxis_Move_02 : DINT;
   p_FiberAxis_Move_02_String : STRING := '0';
   p_FiberGripper_IN : BOOL;
   p_FiberGripper_OUT : BOOL;
   p_FiberLength : DINT;
   p_FiberLength_Initial : DINT;
   p_Free_Running : DINT := 5830001;
   p_HMI_IO_Display : udt_HMI_IO_Desc := (Increment_Page := 1, Increment_OS := 1, Decrement_Page := 1, Decrement_OS := 1, Index := 3, Max_Index := 3, IO_Desc[0].Address := 'VS_063:O:0.0', IO_Desc[0].Description := 'Cassette Release');
   p_HMI_MachineStatus : DINT;
   p_HMI_Message_Active : udt_HMI_Message_Display := (Message.Message := 'Safety Reset Required', Message.Background := 6);
   p_HMI_Message_Sequence_Active : udt_HMI_Message_Display := (Message.Message := 'Waiting for Cassette', Message.Background := 4, Index := 1);
   p_HMI_PLC_Status : udt_Controller_Status := (Controller_Mode := 3, Controller_Status := 12640, Device_Status := 6, Fault_Status := 1, IO_Status := 2, Key_Switch_Status := 3, Minor_Fault := 16);
   p_LED_01 : udt_LED;
   p_LED_02 : udt_LED;
   p_LED_03 : udt_LED;
   p_LED_04 : udt_LED;
   p_LED_Ramp : BOOL;
   p_LED_Ramp_Done : BOOL;
   p_LifeTime_Part_Counter : DINT;
   p_MainAirOkay_IN : BOOL;
   p_MirrorAxis : udt_Zaber_Axis := (Home := 1, ActPos_Step_String := '0', CmdPos_mm := 29.999924, CmdPos_Step_Dint := 241890, CmdPos_Step_String := '241890', Home_String := '/1 3 home$0D', MovAbs_String := '/1 3 move abs ', Return_String := '$0D', Resloution := 0.124023, Jog_Fwd_String := '/1 3 move rel  ', Jog_Rev_String := '/1 3 move rel  -', Jog_Value_mm := 10.0, Jog_Value_Step_Dint := 80630, Jog_Value_Step_String := '80630', Get_Pos_String := '/1 3 get pos$0D', Store_CmdPos_Delay.PRE := 1000, String_Pos_Found := 20, String_Pos_Length := 1, IdlePos := 11, Zero := '0', Get_Pos_Delay.PRE := 1000, Store_CmdPos_Reset_Delay.PRE := 1500);
        .HMI_PB.PB_OS.0   // Go Cmd Pos
        .HMI_PB.PB_OS.2   // Jog Rev
        .HMI_PB.PB_OS.3   // Jog Fwd
        .HMI_PB.PB_OS.4   // Go Home
   p_OkayToProcess : BOOL;
   p_Part_Counter : DINT;
   p_PBLight_Amber_OUT : BOOL := 1;
   p_PBLight_Green_OUT : BOOL;
   p_PBLight_Red_OUT : BOOL;
   p_Sequence : udt_Station_Sequence := (Home := 1, OS := 1);
   p_StackLight_Amber_OUT : BOOL := 1;
   p_StackLight_Green_OUT : BOOL;
   p_StackLight_Red_OUT : BOOL;
   p_StartPB_IN : BOOL;
   p_SyringeAxis : udt_Zaber_Axis := (Home := 1, ActPos_Step_String := '0', CmdPos_mm := 21.248753, CmdPos_Step_Dint := 111542, CmdPos_Step_String := '111542', Home_String := '/1 2 home$0D', MovAbs_String := '/1 2 move abs ', Return_String := '$0D', Resloution := 0.1905, Jog_Fwd_String := '/1 2 move rel  ', Jog_Rev_String := '/1 2 move rel  -', Jog_Value_mm := 5.0, Jog_Value_Step_Dint := 26247, Jog_Value_Step_String := '26247', Get_Pos_String := '/1 2 get pos$0D', Store_CmdPos_Delay.PRE := 1000, String_Pos_Found := 20, String_Pos_Length := 1, IdlePos := 11, Zero := '0', Get_Pos_Delay.PRE := 500, Store_CmdPos_Reset_Delay.PRE := 1500);
        .HMI_PB.PB_OS.0   // Go Cmd Position
        .HMI_PB.PB_OS.2   // Jog Rev
        .HMI_PB.PB_OS.3   // Jog Fwd
        .HMI_PB.PB_OS.4   // Go Home
   p_syringeAxis_pos_found : DINT;
   p_syringeAxis_pos_Length : DINT;
   p_test_Mode : BOOL;
   p_Uptime : String_15 := '0:00:00';
   p_Waiting : BOOL;
   p_Waiting_Time : String_15 := '0:00:00';
   p_WorkLight_OUT : BOOL := 1;
END_VAR
VAR {public}
   p_Alarm : BOOL;
   p_Machine_Control : udt_Machine_Control_V2 := (Message_Index := 16);
END_VAR

ROUTINE A_Main   (* ladder *)
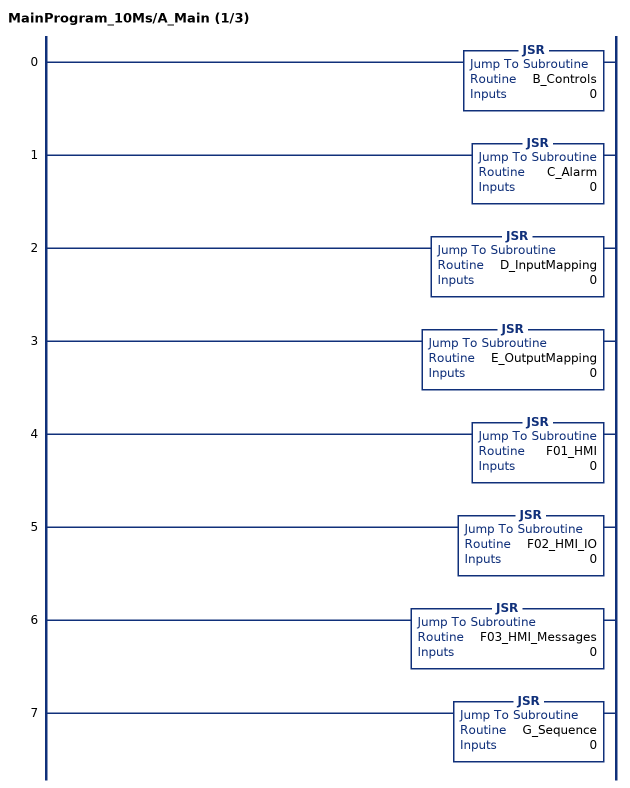
   0: JSR(B_Controls,0);
   1: JSR(C_Alarm,0);
   2: JSR(D_InputMapping,0);
   3: JSR(E_OutputMapping,0);
   4: JSR(F01_HMI,0);
   5: JSR(F02_HMI_IO,0);
   6: JSR(F03_HMI_Messages,0);
   7: JSR(G_Sequence,0);
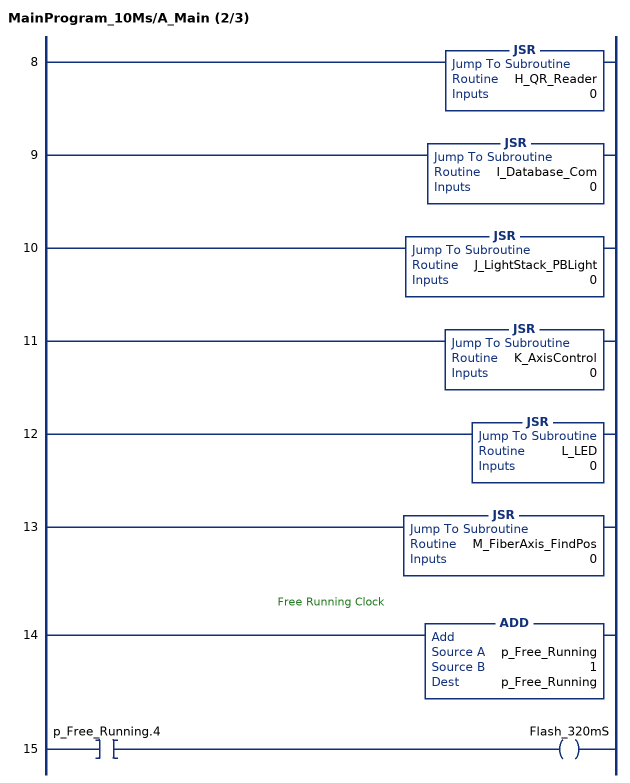
   8: JSR(H_QR_Reader,0);
   9: JSR(I_Database_Com,0);
   10: JSR(J_LightStack_PBLight,0);
   11: JSR(K_AxisControl,0);
   12: JSR(L_LED,0);
   13: JSR(M_FiberAxis_FindPos,0);
   // Free Running Clock
   14: ADD(p_Free_Running,1,p_Free_Running);
   15: XIC(p_Free_Running.4)OTE(Flash_320mS);
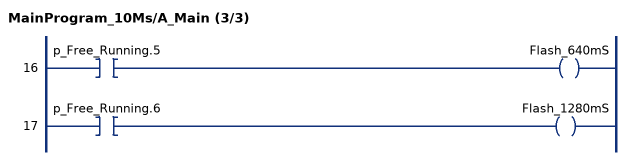
   16: XIC(p_Free_Running.5)OTE(Flash_640mS);
   17: XIC(p_Free_Running.6)OTE(Flash_1280mS);
END_ROUTINE

ROUTINE B_Controls   (* ladder *)
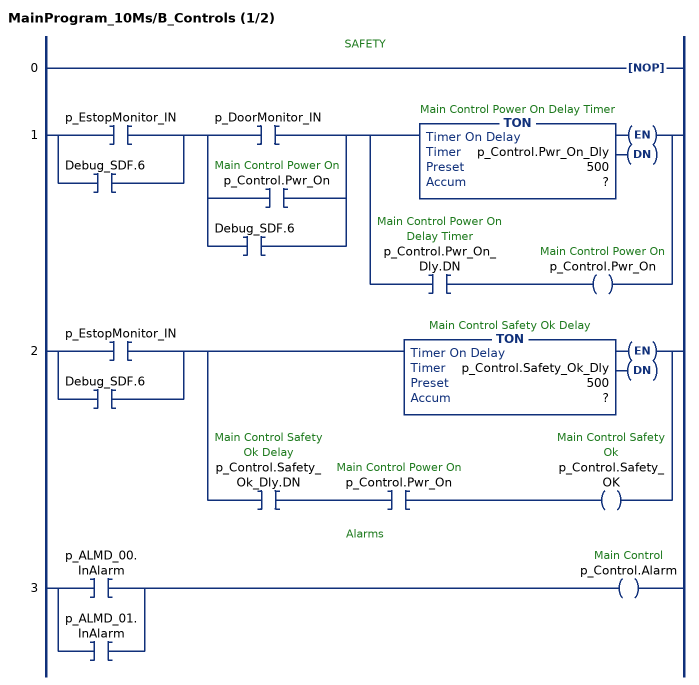
   // SAFETY
   0: NOP();
   1: [XIC(p_EstopMonitor_IN) ,XIC(Debug_SDF.6) ][XIC(p_DoorMonitor_IN) ,XIC(p_Control.Pwr_On) ,XIC(Debug_SDF.6) ][TON(p_Control.Pwr_On_Dly,?,?) ,XIC(p_Control.Pwr_On_Dly.DN) OTE(p_Control.Pwr_On) ];
   2: [XIC(p_EstopMonitor_IN) ,XIC(Debug_SDF.6) ][TON(p_Control.Safety_Ok_Dly,?,?) ,XIC(p_Control.Safety_Ok_Dly.DN) XIC(p_Control.Pwr_On) OTE(p_Control.Safety_OK) ];
   // Alarms
   3: [XIC(p_ALMD_00.InAlarm) ,XIC(p_ALMD_01.InAlarm) ]OTE(p_Control.Alarm);
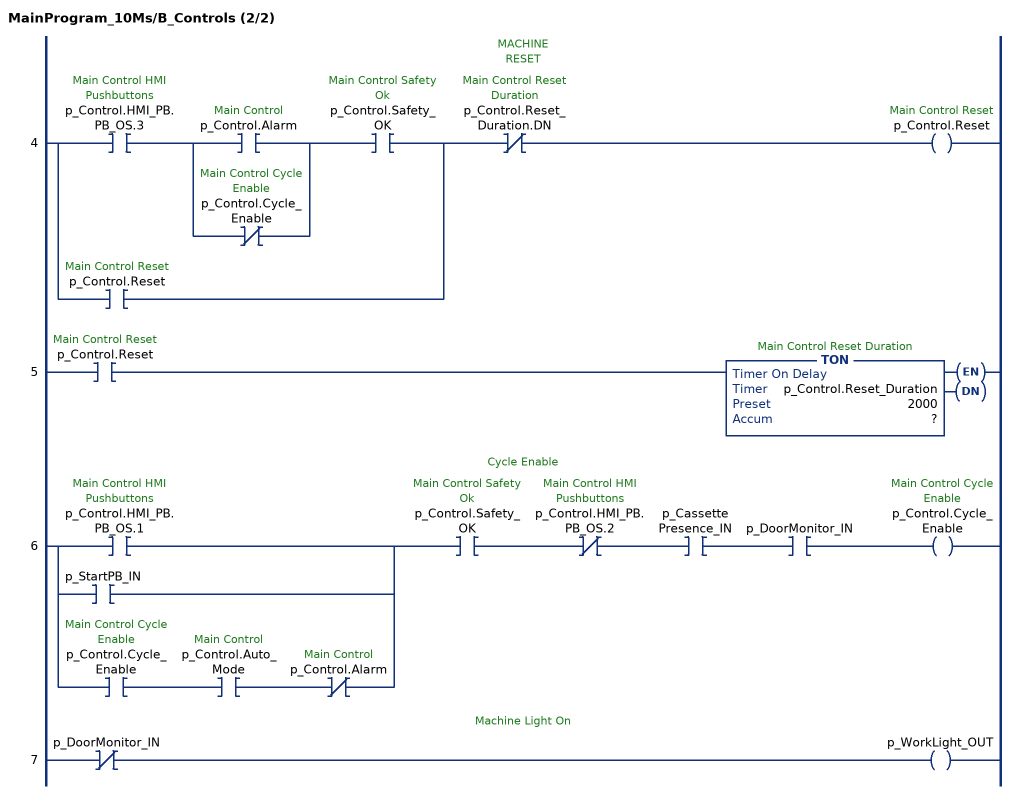
   // MACHINE
   // RESET
   4: [XIC(p_Control.HMI_PB.PB_OS.3) [XIC(p_Control.Alarm) ,XIO(p_Control.Cycle_Enable) ] XIC(p_Control.Safety_OK) ,XIC(p_Control.Reset) ]XIO(p_Control.Reset_Duration.DN)OTE(p_Control.Reset);
   5: XIC(p_Control.Reset)TON(p_Control.Reset_Duration,?,?);
   // Cycle Enable
   6: [XIC(p_Control.HMI_PB.PB_OS.1) ,XIC(p_StartPB_IN) ,XIC(p_Control.Cycle_Enable) XIC(p_Control.Auto_Mode) XIO(p_Control.Alarm) ]XIC(p_Control.Safety_OK)XIO(p_Control.HMI_PB.PB_OS.2)XIC(p_CassettePresence_IN)XIC(p_DoorMonitor_IN)OTE(p_Control.Cycle_Enable);
   // Machine Light On
   7: XIO(p_DoorMonitor_IN)OTE(p_WorkLight_OUT);
END_ROUTINE
